// TwinCAT 3 PLC project Untitled1
// ProgramVersion: 3.1.4024.12
// libraries:
//   Tc2_Standard, * (Beckhoff Automation GmbH)
//   Tc2_System, * (Beckhoff Automation GmbH)
//   Tc3_Module, * (Beckhoff Automation GmbH)
//   VisuSymbols,3.5.10.0,System
// project tree:
//   DUTs/ GEMMA.TcDUT
//   / GlobalTextList.TcGTLO, PlcTask.TcTTO, Visualization Manager.TcVMO (not stored)
//   POUs/ FB_Clock.TcPOU, FB_Controller.TcPOU, FB_Director.TcPOU, FB_F1Production_SFC.TcPOU, FB_Discharger_SFC.TcPOU, FB_Discharger_ST.TcPOU, FB_Object_Template_SFC.TcPOU, FB_Object_Template_ST.TcPOU, FB_Panel.TcPOU, FB_Restoration_SFC.TcPOU, MAIN.TcPOU
//   VISUs/ Visualization.TcVIS
// real-time tasks:
//   TASK PlcTask: cycle T#10ms, priority 20, ADS port 350

CONFIGURATION Untitled1
    RESOURCE PLC ON TwinCAT3
        TASK PlcTask(INTERVAL := T#10ms, PRIORITY := 20);
        PROGRAM MAIN WITH PlcTask : MAIN;
    END_RESOURCE
END_CONFIGURATION

// ---- DUTs/GEMMA.TcDUT
TYPE GEMMA :
(
	  (* Modes de la Guia de Estudio de los Modes de Marcha y Parada *)
    (* [Modes du Guide d'Etude des Modes de Marche et d'Arrêt] *)
    (* [Modes of Study Guide of the Modes of Operating and Stopping] *)

    (* Procedimientos de parada [les procédures d'arrets/stop procedures] *)
    A1ParadaInicial, (*  0: parada en el estado inicial
               [arrêt dans etat initial] 
               [stopped in the initial state] *)
    A2ParaFinCiclo, (*  1: parada solicitada a final de ciclo
               [arret demandé en fin de cycle] 
               [requested end cycle stop] *)
    A3ParadaEstado, (*  2: parada solicitada en un estado determinado
               [arret demande dans etat determine] 
               [requested particular state stop] *)
    A4ParadaObtenida, (*  3: parada obtenida
               [arret obtenu] 
               [obteined stop] *)
    A5PreparandoTrasFallo, (*  4: preparacion para la recuperacion del fallo
               [preparation pour remise en route apres defaillance] 
               [preparation for the recovery of the Fail] *)
    A6Inicializando, (*  5: situando la PO en el estado inicial
               [mise PO dans état initial] 
               [set the PO in initial state] *)
    A7SituandoEstado, (*  6: situando la PO en un estado determinado
               [mise PO dans état déterminé]
               [set the PO in a certain state] *)

    (* Procedimientos de funcionamiento [les procédures de fonctionnement/operating procedures] *)
    F1ProduccionNormal, (*  7: produccion normal
               [production normale] 
               [normal operation] *)
    F2SecuenciaPreparacion, (*  8: secuencia de preparacion
               [marche de preparation] 
               [preparation sequence] *)
    F3SecuenciaFinalizacion, (*  9: secuencia de finalizacion
               [marche de cloture] 
               [ending sequence] *)
    F4VerificacionSinOrden, (* 10: verificacion en desorden
               [marche de verification dans le desordre] 
               [verification with no order] *)
    F5VerificacionOrdenada, (* 11: verificacion en orden
               [marche de verification dans l'ordre] 
               [verification whit order] *)
    F6Probando, (* 12: prueba
               [marche de test] 
               [test] *)

    (* Procedimientos de fallo [les procédures en défaillances] *)
    D1ParadaEmergencia, (* 13: parada de emergencia
               [arret d'urgence] 
               [emergency stop] *)
    D2TratamientoFallos, (* 14: diagnostico y/o tratamiento de los fallos
               [diagnostic et/ou traitement de la défaillance] 
               [diagnosis and/or treatment of Fails] *)
    D3ProducirConFallos  (* 15: produccion a pesar de los fallos
               [production tout de même] 
               [production despite the Fails] *)
);
END_TYPE

// ---- POUs/MAIN.TcPOU
PROGRAM MAIN
VAR
	Controller: FB_Controller;
END_VAR

Controller();

END_PROGRAM

// ---- POUs/FB_Controller.TcPOU
FUNCTION_BLOCK FB_Controller EXTENDS FB_Object_Template_ST
VAR_INPUT
	//Discharger
	Tray_1 : BOOL; 
	Tray_2 : BOOL;
END_VAR
VAR_OUTPUT
	Fail : BOOL;
END_VAR
VAR
	Director   : FB_Director;
	Discharger : FB_Discharger_ST;
	Production : FB_F1Production_SFC;
	Panel      : FB_Panel;
	End: BOOL;
END_VAR

IC := Discharger.IC;
End := Production.Done;
Director(Emergency :=  Panel.Emergency,
		 Endbatch := Production.Done,
		 End := End,
		 Fail := Fail,
		 Go := Panel.Go,
		 Manual := Panel.Manual,
		 Reboot := Panel.Reboot,
		 Restore := IC,
		 Stop := Panel.Stop
		 );

Production(Execute := (Director.Mode=F1ProduccionNormal), 
			Ack :=Ack,
			SFCReset:=Reset,
			SFCPause :=Pause,
			IC:=IC,
			Discharger_Done:=Discharger.Done,
			);
			
		 
Panel (Mode := Director.Mode);

Discharger(Execute:=Production.Discharger_Execute,
			Ack:=Production.Discharger_Ack,
			Reset:=Reset,
			Pause:=Pause,
			Tray_1:=Tray_1,
			Tray_2:=Tray_2
			);

END_FUNCTION_BLOCK

// ---- POUs/FB_Object_Template_ST.TcPOU
FUNCTION_BLOCK FB_Object_Template_ST
VAR_INPUT
	// Control variables
	Execute: BOOL;
	Ack: BOOL;
	Reset: BOOL; 
	Pause: BOOL;
	// Physical variables
	
END_VAR
VAR_OUTPUT
	//Control variables
	Ready: BOOL;
	Done: BOOL;
	//Physical Variables
	
END_VAR
VAR
	// Initial conditions
	IC: BOOL := TRUE;
END_VAR

END_FUNCTION_BLOCK

// ---- POUs/FB_Director.TcPOU
FUNCTION_BLOCK FB_Director
VAR_INPUT
	//Panel Buttons
	Emergency :BOOL; //seta
	EndBatch  :BOOL;
	End		  :BOOL;
	Fail  	  :BOOL;
	Go        :BOOL; //marcha
	Manual 	  :BOOL; //manual
	Reboot 	  :BOOL;
	Restore   :BOOL;
	Stop      :BOOL; //parada

END_VAR
VAR_OUTPUT
	Mode : GEMMA := GEMMA.A6Inicializando;
	Pause : BOOL;
	Production : BOOL;
		
END_VAR
VAR
	ModeAns: GEMMA;
END_VAR

(* Define output commands*)
Pause := (Mode = A3ParadaEstado) 
		 OR (Mode = A4ParadaObtenida) 
		 OR (Mode = A5PreparandoTrasFallo)
		 OR (Mode = D1ParadaEmergencia) 
		 OR (Mode = D2TratamientoFallos);
Production := (Mode = A2ParaFinCiclo)
		   OR (Mode = A3ParadaEstado)
		   OR (Mode = F1ProduccionNormal)
		   OR (Mode = F2SecuenciaPreparacion)
		   OR (Mode = F3SecuenciaFinalizacion)
		   OR (Mode = F5VerificacionOrdenada)
		   OR (Mode = F6Probando)
		   OR (Mode = D3ProducirConFallos);
(* Choose mode *)

IF Reboot THEN
	Mode := A6Inicializando;
ELSIF Emergency THEN
	Mode := D1ParadaEmergencia;
END_IF

CASE Mode OF
	// ARRÈT 
	A1ParadaInicial:
	IF Manual THEN
		Mode := F4VerificacionSinOrden;
	ELSIF Go THEN
		Mode := F2SecuenciaPreparacion;
	END_IF
	
	A2ParaFinCiclo:
	IF Fail THEN
		ModeAns := A2ParaFinCiclo;
		Mode 	:= D2TratamientoFallos;
	ELSIF EndBatch THEN
		Mode := A1ParadaInicial;
	END_IF
	
	A5PreparandoTrasFallo: 
	IF Go THEN
		Mode := A1ParadaInicial;
	ELSIF Stop THEN
		Mode := A6Inicializando;
	END_IF
	
	A6Inicializando:
	IF Restore THEN
		Mode := A1ParadaInicial;
	ELSIF Manual THEN
		Mode := F4VerificacionSinOrden;
	END_IF
	
	// Fonctionnement
	F1ProduccionNormal: 
	IF Fail THEN
		ModeAns := A2ParaFinCiclo;
		Mode := D2TratamientoFallos;
	ELSIF EndBatch THEN
		Mode := F3SecuenciaFinalizacion;
	ELSIF Stop THEN
		Mode := A2ParaFinCiclo;
	END_IF
	
	F3SecuenciaFinalizacion: 
	IF End THEN
		Mode := A1ParadaInicial;
	END_IF
	
	F4VerificacionSinOrden:
	IF NOT Manual THEN
		Mode := A6Inicializando;
	ELSIF Fail THEN
		ModeAns := A2ParaFinCiclo;
		Mode := D2TratamientoFallos;
	END_IF
	
	// Défail
	D1ParadaEmergencia :
	IF NOT Emergency THEN
		Mode := A6Inicializando;
	END_IF
	
	D2TratamientoFallos:
	IF NOT Fail THEN
		Mode := A5PreparandoTrasFallo;
	END_IF
END_CASE

END_FUNCTION_BLOCK

// ---- POUs/FB_Discharger_ST.TcPOU
FUNCTION_BLOCK FB_Discharger_ST EXTENDS FB_Object_Template_ST
VAR_INPUT
	Tray_1: BOOL; 
	Tray_2: BOOL;
	dcha_1 AT %I*: BOOL;
	dcha_2 AT %I*: BOOL;
	izda_1 AT %I*: BOOL;
	izda_2 AT %I*: BOOL;
	arriba AT %I*: BOOL;
	abajo  AT %I*: BOOL;
	cogido AT %I*: BOOL;
END_VAR
VAR_OUTPUT
	avanza_1 AT %Q*: BOOL;
	avanza_2 AT %Q*: BOOL;
	baja	 AT %Q*: BOOL;
	coge 	 AT %Q*: BOOL;
	Fail : BOOL;
	Timer : TON;
END_VAR
VAR
	Discharger : FB_Discharger_SFC;
END_VAR

//Define initial conditions
IC := izda_1 AND izda_2 AND arriba AND NOT cogido;
Fail := F_Fail(Timer);
//Declare module
Discharger(Execute:=Execute,
		   Ack:=Ack,
		   SFCReset:=Reset,
		   SFCPause:=Pause,
		   IC:=IC,
		   Tray_1:=Tray_1,
		   Tray_2:=Tray_2,
		   dcha_1:=dcha_1,
		   dcha_2:=dcha_2,
		   izda_1:=izda_1,
		   izda_2:=izda_2,
		   arriba:=arriba,
		   abajo:=abajo,
		   cogido:=cogido,
Restore := _REFACTOR_
);
		   
//Declare module actuators
Ready := Discharger.Ready;
Done := Discharger.Done;
avanza_1 := Discharger.avanza_1;
avanza_2 := Discharger.avanza_2;
baja := Discharger.baja;
coge := Discharger.coge;

METHOD F_Fail : BOOL
VAR_INPUT
	Timer : TON;
END_VAR
VAR
	NumError : UDINT;
	Message  : STRING;
END_VAR
F_Fail := FALSE;
END_METHOD

END_FUNCTION_BLOCK

// ---- POUs/FB_Discharger_SFC.TcPOU
FUNCTION_BLOCK FB_Discharger_SFC EXTENDS FB_Object_Template_SFC
VAR_INPUT
	Tray_1: BOOL;
	Tray_2: BOOL;
	dcha_1: BOOL;
	dcha_2: BOOL;
	izda_1: BOOL;
	izda_2: BOOL;
	arriba: BOOL;
	abajo: BOOL;
	cogido: BOOL;
	Restore: BOOL;
END_VAR
VAR_OUTPUT
	avanza_1: BOOL;
	avanza_2: BOOL;
	baja: BOOL;
	coge: BOOL;
END_VAR
VAR
END_VAR

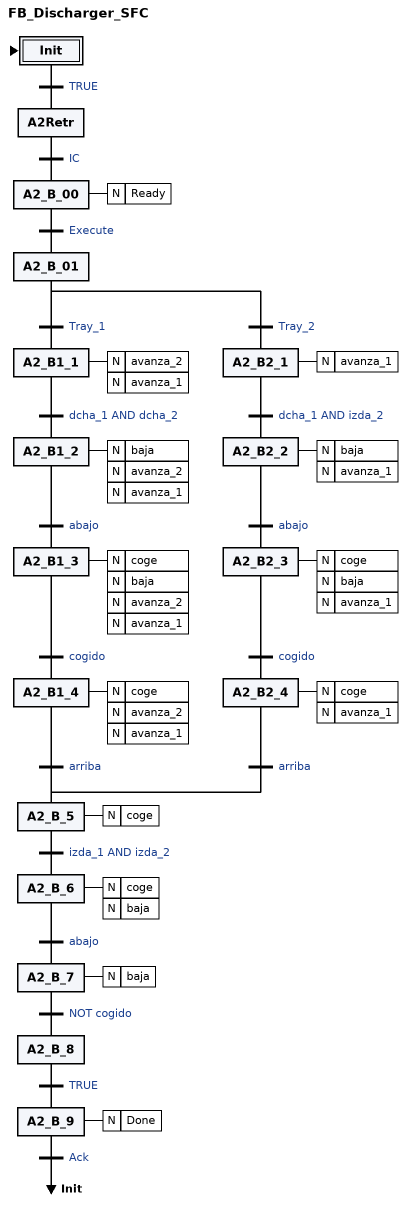
INITIAL_STEP Init:
END_STEP
TRANSITION FROM Init TO A2Retr
    := TRUE;
END_TRANSITION
STEP A2Retr:
END_STEP
TRANSITION FROM A2Retr TO A2_B_00
    := IC;
END_TRANSITION
STEP A2_B_00:
    Ready(N);
END_STEP
TRANSITION FROM A2_B_00 TO A2_B_01
    := Execute;
END_TRANSITION
STEP A2_B_01:
END_STEP
TRANSITION FROM A2_B_01 TO A2_B1_1
    := Tray_1;
END_TRANSITION
STEP A2_B1_1:
    avanza_2(N);
    avanza_1(N);
END_STEP
TRANSITION FROM A2_B1_1 TO A2_B1_2
    := dcha_1 AND dcha_2;
END_TRANSITION
STEP A2_B1_2:
    baja(N);
    avanza_2(N);
    avanza_1(N);
END_STEP
TRANSITION FROM A2_B1_2 TO A2_B1_3
    := abajo;
END_TRANSITION
STEP A2_B1_3:
    coge(N);
    baja(N);
    avanza_2(N);
    avanza_1(N);
END_STEP
TRANSITION FROM A2_B1_3 TO A2_B1_4
    := cogido;
END_TRANSITION
STEP A2_B1_4:
    coge(N);
    avanza_2(N);
    avanza_1(N);
END_STEP
TRANSITION FROM A2_B1_4 TO A2_B_5
    := arriba;
END_TRANSITION
TRANSITION FROM A2_B_01 TO A2_B2_1
    := Tray_2;
END_TRANSITION
STEP A2_B2_1:
    avanza_1(N);
END_STEP
TRANSITION FROM A2_B2_1 TO A2_B2_2
    := dcha_1 AND izda_2;
END_TRANSITION
STEP A2_B2_2:
    baja(N);
    avanza_1(N);
END_STEP
TRANSITION FROM A2_B2_2 TO A2_B2_3
    := abajo;
END_TRANSITION
STEP A2_B2_3:
    coge(N);
    baja(N);
    avanza_1(N);
END_STEP
TRANSITION FROM A2_B2_3 TO A2_B2_4
    := cogido;
END_TRANSITION
STEP A2_B2_4:
    coge(N);
    avanza_1(N);
END_STEP
TRANSITION FROM A2_B2_4 TO A2_B_5
    := arriba;
END_TRANSITION
STEP A2_B_5:
    coge(N);
END_STEP
TRANSITION FROM A2_B_5 TO A2_B_6
    := izda_1 AND izda_2;
END_TRANSITION
STEP A2_B_6:
    coge(N);
    baja(N);
END_STEP
TRANSITION FROM A2_B_6 TO A2_B_7
    := abajo;
END_TRANSITION
STEP A2_B_7:
    baja(N);
END_STEP
TRANSITION FROM A2_B_7 TO A2_B_8
    := NOT cogido;
END_TRANSITION
STEP A2_B_8:
END_STEP
TRANSITION FROM A2_B_8 TO A2_B_9
    := TRUE;
END_TRANSITION
STEP A2_B_9:
    Done(N);
END_STEP
TRANSITION FROM A2_B_9 TO Init
    := Ack;
END_TRANSITION

END_FUNCTION_BLOCK

// ---- POUs/FB_Object_Template_SFC.TcPOU
FUNCTION_BLOCK FB_Object_Template_SFC
VAR_INPUT
	// Control variables
	Execute: BOOL;
	Ack: BOOL;
	SFCReset: BOOL; 
	SFCPause: BOOL;
	IC: BOOL;
	// Physical variables
END_VAR
VAR_OUTPUT
	//Control variables
	Ready: BOOL;
	Done: BOOL;
	//Physical Variables
END_VAR
VAR
END_VAR

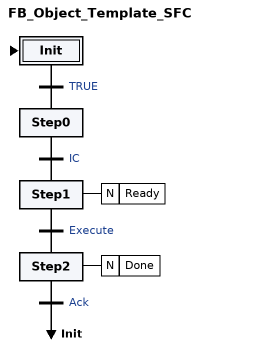
INITIAL_STEP Init:
END_STEP
TRANSITION FROM Init TO Step0
    := TRUE;
END_TRANSITION
STEP Step0:
END_STEP
TRANSITION FROM Step0 TO Step1
    := IC;
END_TRANSITION
STEP Step1:
    Ready(N);
END_STEP
TRANSITION FROM Step1 TO Step2
    := Execute;
END_TRANSITION
STEP Step2:
    Done(N);
END_STEP
TRANSITION FROM Step2 TO Init
    := Ack;
END_TRANSITION

END_FUNCTION_BLOCK

// ---- POUs/FB_F1Production_SFC.TcPOU
FUNCTION_BLOCK FB_F1Production_SFC EXTENDS FB_Object_Template_SFC
VAR_INPUT
//Discharger
	Discharger_Ready: BOOL;
	Discharger_Done: BOOL;
END_VAR
VAR_OUTPUT
	//Discharger
	Discharger_Execute: BOOL;
	Discharger_Ack: BOOL;
END_VAR
VAR
END_VAR

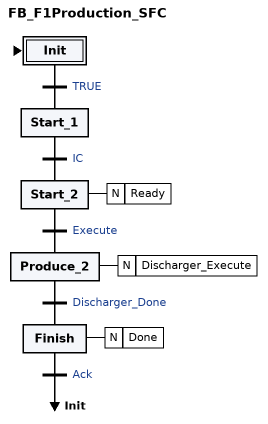
INITIAL_STEP Init:
END_STEP
TRANSITION FROM Init TO Start_1
    := TRUE;
END_TRANSITION
STEP Start_1:
END_STEP
TRANSITION FROM Start_1 TO Start_2
    := IC;
END_TRANSITION
STEP Start_2:
    Ready(N);
END_STEP
TRANSITION FROM Start_2 TO Produce_2
    := Execute;
END_TRANSITION
STEP Produce_2:
    Discharger_Execute(N);
END_STEP
TRANSITION FROM Produce_2 TO Finish
    := Discharger_Done;
END_TRANSITION
STEP Finish:
    Done(N);
END_STEP
TRANSITION FROM Finish TO Init
    := Ack;
END_TRANSITION

END_FUNCTION_BLOCK

// ---- POUs/FB_Panel.TcPOU
FUNCTION_BLOCK FB_Panel
VAR_INPUT
   Mode: GEMMA;
   Restart_Time: TIME := T#3S;

END_VAR
VAR_OUTPUT
	Emergency: BOOL;
	Go:     BOOL;
	Manual:     BOOL;
    Stop:       BOOL;
    Reboot:   BOOL; (* Restablece situacion inicial *)
    Restore:   BOOL; (* Restaura condiciones iniciales *)
END_VAR
VAR
    (* Bloques funcionales *)
    CLK: FB_Clock;
    Trig_PGo: R_TRIG;
    TmpReinicio: TON;

    (* Entradas *)
    PEmergency AT %I*: BOOL; (* Pulsador de parada de emergencia [EMERGENCY STOP] *)
    PGo AT %I*: BOOL; (* Pulsador de marcha [START] *)
    PStop AT %I*: BOOL := TRUE; (* Pulsador de parada [STOP] *)
    PManual AT %I*: BOOL; (* Selector de Mode AUTO/MAN [AUTO/MAN] *)

    (* Salidas *)
    Red_Lamp    AT %Q*: BOOL; (* Lampara de alarma [ALARM] *)
	Yellow_Lamp AT %Q*: BOOL; (* Lampara de alarma [ALARM] *)
	Green_Lamp  AT %Q*: BOOL; (* Lampara de alarma [ALARM] *)
END_VAR

(* PARAMETROS DE SALIDA *)
Emergency:= PEmergency;
Manual := PManual;
Reboot := TmpReinicio.Q;
Restore := PGo;
Go := Trig_PGo.Q;
Stop := PStop;

(* ACCIONES *)
Red_Lamp := (Mode = F3SecuenciaFinalizacion) OR (((Mode = D1ParadaEmergencia) OR (Mode = D2TratamientoFallos) OR (Mode = F2SecuenciaPreparacion)) AND CLK.Q);
Yellow_Lamp := ((Mode = A6Inicializando) OR (Mode = D1ParadaEmergencia) OR (Mode = D2TratamientoFallos)) AND CLK.Q;
Green_Lamp := ((Mode = A2ParaFinCiclo) OR (Mode = F1ProduccionNormal) OR (Mode = F2SecuenciaPreparacion) OR (Mode = F3SecuenciaFinalizacion)) OR ((Mode = A1ParadaInicial) AND CLK.Q);

(* BLOQUES FUNCIONALES *)
CLK();

Trig_PGo(CLK := PGo);

TmpReinicio(
    IN := PGo AND NOT PStop,
	PT := Restart_Time
    );

END_FUNCTION_BLOCK

// ---- POUs/FB_Clock.TcPOU
FUNCTION_BLOCK FB_Clock
(*
Copyright (c) 2009-2017 victortorreslopez
GNU General Public License
*)
VAR_INPUT
  EN: BOOL := TRUE;	(* ENabled *)
  PT: TIME := T#500ms; (* Semicycle time *)
END_VAR
VAR_OUTPUT
  ET: TIME; (* Elapsed time *)
  Q: BOOL; (* Square wave *)
END_VAR
VAR
  Timer: TON; (* Auto-pilot timer *)
END_VAR

(* OUTPUT FUNCTION *)
IF Timer.Q THEN
  Q := NOT Q;
END_IF

(* FUNCTION BLOCKS *)
Timer(IN := EN AND NOT Timer.Q, PT := PT, ET => ET);

END_FUNCTION_BLOCK

// ---- POUs/FB_Restoration_SFC.TcPOU
FUNCTION_BLOCK FB_Restoration_SFC EXTENDS FB_Object_Template_ST
VAR_INPUT
END_VAR
VAR_OUTPUT
END_VAR
VAR
END_VAR

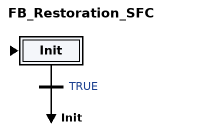
INITIAL_STEP Init:
END_STEP
TRANSITION FROM Init TO Init
    := TRUE;
END_TRANSITION

END_FUNCTION_BLOCK

// ---- GlobalTextList.TcGTLO
TEXTLIST GlobalTextList
  85 = 'abajo'
  971 = 'arriba'
  417 = 'cogido'
  651 = 'dcha_1'
  189 = 'dcha_2'
  370 = 'Execute'
  734 = 'izda_1'
  121 = 'izda_2'
  251 = 'Pause'
  530 = 'Reset'
  933 = 'Tray 1'
  492 = 'Tray 2'
END_TEXTLIST

// ---- VISUs/Visualization.TcVIS
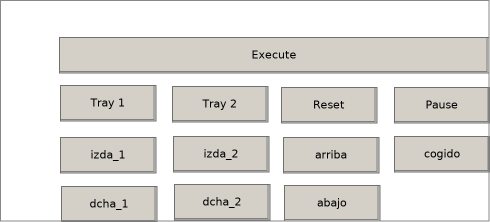
VISUALIZATION Visualization  // 490x222
    Button (59,37 430x36), "Execute"
        tap MAIN.Controller.Execute
    Button (60,85 96x36), "Tray 1"
        tap MAIN.Controller.Tray_1
    Button (172,86 96x36), "Tray 2"
        tap MAIN.Controller.Tray_2
    Button (60,137 96x36), "izda_1"
        toggle MAIN.Controller.Discharger.izda_1
    Button (173,136 96x36), "izda_2"
        toggle MAIN.Controller.Discharger.izda_2
    Button (283,137 96x36), "arriba"
        toggle MAIN.Controller.Discharger.arriba
    Button (394,136 96x36), "cogido"
        toggle MAIN.Controller.Discharger.cogido
    Button (281,87 96x36), "Reset"
        tap MAIN.Controller.Reset
    Button (394,87 96x36), "Pause"
        tap MAIN.Controller.Pause
    Button (61,186 96x36), "dcha_1"
        toggle MAIN.Controller.Discharger.dcha_1
    Button (174,184 96x36), "dcha_2"
        toggle MAIN.Controller.Discharger.dcha_2
    Button (284,185 96x36), "abajo"
        toggle MAIN.Controller.Discharger.abajo
END_VISUALIZATION
